TYPE DigitalInputBase_50022E7B :
STRUCT
END_STRUCT
END_TYPE

(* stored: Version 1.2.0.0, ProductVersion 3.1.4024.9
   DUT DigitalInputBase_50022E7B: Id {b72c4a39-0cc4-4cea-88bd-208dd582ba5d} *)
